(* CoDeSys 2.3.9.47 project: lab_4.pro *)
(* Libraries: STANDARD.LIB 5.6.98 11:03:02 *)

(* Task configuration *)
TASK Standard (PRIORITY := 0, INTERVAL := T#10ms);
	MAIN
END_TASK

(* Global variable list: Global_Variables *)
VAR_GLOBAL
	(*Global used Time [sec]*)
	t_global : REAL;
END_VAR

(* Data type *)
TYPE T_STATE :
(
	STATE_IDLE := 0,
	STATE_RISE1:= 1,
	STATE_RISE2:= 2,
	STATE_FALL1:= 3,
	STATE_FALL2:= 4
);
END_TYPE

(* POU MAIN, ST *)
PROGRAM MAIN
VAR
	(*System Block*)
	var_int		:Integrator;
	var_lp		: LowpassFilter;	

	(*Function Input Parameters*)
	mini_sqr	:REAL := -2;
	maxi_sqr	:REAL := +2;
	tau			:REAL := 0.1;
	
	(*Function Output Signals*)
	sigOut_int	: REAL := 0;
	sigOut_sqr	: REAL := 0;
	sigOut_lp	: REAL := 0;
END_VAR
(*Initialize Function Blocks*)
var_int();
var_lp();

(*Square Wave*)
sigOut_sqr := SquareSignal(t_global, mini_sqr, maxi_sqr);

(*Call Integrator*)
var_int.e_k := sigOut_sqr;
(*Write Integral Value in Variable*)
sigOut_int := var_int.u_k;

(*Call Lowpass Filter*)
var_lp.x_k	:= sigOut_sqr;
(*Write Lowpassed in Variable*)
sigOut_lp	:= var_lp.y_k;

(*Increment global Time*)
t_global := t_global + 0.01;
END_PROGRAM

(* POU Integrator, ST *)
FUNCTION_BLOCK Integrator
VAR_INPUT
	e_k		: REAL ;
END_VAR
VAR_OUTPUT
	u_k	: REAL ;
END_VAR
VAR
	u_k_1	: REAL;
	e_k_1	: REAL;
	T		: REAL := 0;
	T_leave	: REAL := 0;
END_VAR
(*Calculate Time Gap*)
IF t_global = 0 THEN
	T := 0.01;
ELSE
	T := t_global - T_leave;
END_IF

(*Trapeze Approximation*)
Integrator.u_k := u_k_1 + (e_k + e_k_1)*T/2;


(*Actualize later used Variables*)
e_k_1 := e_k;
u_k_1 := u_k;
T_leave := t_global;
END_FUNCTION_BLOCK

(* POU LowpassFilter, ST *)
FUNCTION_BLOCK LowpassFilter
VAR_INPUT
	x_k		: REAL;
	tau		: REAL;
END_VAR
VAR_OUTPUT
	y_k		: REAL;
END_VAR
VAR
	y_k_1	: REAL;
	T		: REAL;
	T_leave : REAL;
	p	 	: REAL;
	q		: REAL;
END_VAR
(*Calculate Time Gap*)
IF t_global = 0 THEN
	T := 0.01;
ELSE
	T := t_global - T_leave;
END_IF

(*Calculate Gains*)
q	:= tau/(T+tau);
p	:= T/(T+tau);


(*Calculate Output*) 
LowpassFilter.y_k := p*x_k + q*y_k_1;


(*Actualize Later used Variables*)
y_k_1 := y_k;
T_leave := t_global;
END_FUNCTION_BLOCK

(* POU SquareSignal, ST *)
FUNCTION SquareSignal : REAL
VAR_INPUT
	t	:	REAL;		(*Input Time*)
	mini:	REAL;		(*Minimum Value*)
	maxi:	REAL;		(*Maximum Value*)
END_VAR
VAR
	w		:	REAL := 1; 	(*Frequency*)
	offs	:	REAL := 0;	(*Offset*)
	curr_sin:	REAL ;		(*Current Sine Wave*)
END_VAR
(*Generate Square-Wave*)

curr_sin := SIN(w*t);

IF curr_sin > 0 THEN
	SquareSignal := maxi + offs;
ELSE
	SquareSignal := mini + offs;
END_IF
END_FUNCTION

(* POU DoubleEdgeDetector, ST *)
FUNCTION_BLOCK DoubleEdgeDetector
VAR_INPUT
	(*Input Signal*)
	sig_in 		: BOOL ;
	(*Timer Count*)
	t			: REAL ;
	(*Idle Time*)
	Ti			: REAL  ;
END_VAR
VAR_OUTPUT
	fall		: BOOL ;
	falls		: BOOL ;	
	rise		: BOOL ;
	rises		: BOOL ;
	(*Timer Commands*)
	timer_ON	: BOOL ;
END_VAR
VAR
	c_state		: T_STATE := STATE_IDLE;
	prev_sig	: BOOL := FALSE;
	edgeRise	: BOOL := FALSE;
	edgeFall	: BOOL := FALSE;
	TOF			: BOOL := FALSE;
END_VAR
(*Reset Outputs*)
DoubleEdgeDetector.fall		:= FALSE ;
DoubleEdgeDetector.falls		:= FALSE ;
DoubleEdgeDetector.rise		:= FALSE ;
DoubleEdgeDetector.rises		:= FALSE ;

(*Check Timer Overflow*)
IF (t > Ti) THEN
	TOF := TRUE;
ELSE
	TOF := FALSE;
END_IF

(*Check Edge*)
IF (prev_sig = sig_in) THEN
	(*Reset Edge*)
	edgeFall := FALSE;
	edgeRise := FALSE;
ELSIF (prev_sig = TRUE) AND (sig_in = FALSE) THEN
	(*Falling Edge*)
	edgeFall := TRUE;
	edgeRise := FALSE;
ELSIF (prev_sig = FALSE) AND (sig_in = TRUE) THEN
	(*Rising Edge*)
	edgeFall := FALSE;
	edgeRise := TRUE;
END_IF

(*Set current Signal = previous Signal*)
prev_sig := sig_in;

(*Final State Machine Implementation*)
CASE c_state OF
	STATE_IDLE:
		(**)
		IF edgeRise = TRUE THEN
			c_state := STATE_RISE1;
		ELSIF edgeFall = TRUE THEN
			c_state := STATE_FALL1;
		ELSE
			c_state := STATE_IDLE;
		END_IF

	STATE_RISE1:
		(*Start Timer*)
		DoubleEdgeDetector.timer_ON := TRUE;
		(**)
		IF TOF = TRUE THEN
			DoubleEdgeDetector.timer_ON := FALSE;
			DoubleEdgeDetector.rise 	:= TRUE;
			c_state := STATE_IDLE;
		ELSIF edgeRise THEN
			c_state := STATE_RISE2;
		ELSE
			c_state := STATE_RISE1;
		END_IF

	STATE_RISE2:
		(**)
		DoubleEdgeDetector.rises 	:= TRUE;
		c_state := STATE_IDLE;
		
	STATE_FALL1:
		(*Start Timer*)
		DoubleEdgeDetector.timer_ON := TRUE;
		(**)
		IF TOF = TRUE THEN
			DoubleEdgeDetector.timer_ON := FALSE;
			DoubleEdgeDetector.fall 	:= TRUE;
			c_state := STATE_IDLE;
		ELSIF edgeFall THEN
			c_state := STATE_FALL2;
		ELSE
			c_state := STATE_FALL1;
		END_IF

	STATE_FALL2:
		(**)
		DoubleEdgeDetector.falls 	:= TRUE;
		c_state := STATE_IDLE;

	ELSE
		c_state := STATE_IDLE;
END_CASE;
END_FUNCTION_BLOCK

(* POU PWMSignal, ST *)
FUNCTION PWMSignal : REAL
VAR_INPUT
	t	:	REAL;		(*Input Time*)
	dc	:	REAL;		(*Input Duty Cicle*)
	per	:	REAL;		(*Input Period*)
END_VAR
VAR
	pi		:	REAL := 3.14159;
	w		:	REAL ;	(*Frequency*)
	th		:	REAL ;
	curr_sin:	REAL ;	(*Current Sine Wave*)
END_VAR
(*Generate PWM*)

(*Calculate Frequency using Period*)
w := (2*pi)/(per);
(*Generate Reference Wave*)
curr_sin := 0.5*SIN(w*t)+0.5;
(*Calculate Threshold*)
th := 1-((dc)/(100));
(*Check validity of Input Duty Call*)
IF (dc <= 0) OR (dc > 100) THEN
	PWMSignal := 0;
ELSE
(*Compare Reference Wave to Threshold*)
IF curr_sin > th THEN
	PWMSignal := 1;
ELSE
	PWMSignal := 0;
END_IF
END_IF
END_FUNCTION

(* POU SecondOrderLag, ST *)
FUNCTION_BLOCK SecondOrderLag
VAR_INPUT
	d	: REAL;
	w0	: REAL;
	x_k	: REAL;
END_VAR
VAR_OUTPUT
	y_k	: REAL;
END_VAR
VAR
	y_k_1	: REAL;
	y_k_2	: REAL;
	T		: REAL;
	T_leave : REAL;
	(*Coefficients*)
	a		: REAL;
	b		: REAL;
	c		: REAL;

END_VAR
(*Calculate Time Gap*)
IF t_global = 0 THEN
	T := 0.001;
ELSE
	T := t_global - T_leave;
END_IF

(*Coefficients*)
a := (1/EXPT(T,2))+((1/T)*2*d*w0)+(EXPT(w0,2));
b := (2/EXPT(T,2))+((1/T)*2*w0);
c := 1/EXPT(T,2);

(*Calculate Output*)
SecondOrderLag.y_k := (1/a)*((EXPT(w0,2))*x_k - b*y_k_1 - c*y_k_2);

(*Actualize Later used Variables*)
y_k_1 := y_k;
y_k_2 := y_k_1;
T_leave := t_global;
END_FUNCTION_BLOCK

(* POU SinusFunction, ST *)
FUNCTION SinusFunction : REAL
VAR_INPUT
	t	:	REAL;		(*Input Time*)
END_VAR
VAR
	w	:	REAL := 1; 	(*Frequency*)
	A	:	REAL := 1;	(*Amplitude*)
	offs:	REAL := 0;	(*Offset*)
END_VAR
(*Generate Sine-Wave*)
SinusFunction := A*SIN(w*t) + offs;
END_FUNCTION
